FUNCTION_BLOCK FB_ERROR_CODE
VAR_INPUT
END_VAR
VAR_OUTPUT
END_VAR
VAR
END_VAR

END_FUNCTION_BLOCK

(* stored: Version 1.1.0.1, ProductVersion 3.1.4024.12
   POU FB_ERROR_CODE: Id {582f2577-f0f5-466d-8f42-319308e7f4ba}, SpecialFunc None *)
